FUNCTION_BLOCK FB_Generator_Random
VAR_INPUT
END_VAR
VAR_OUTPUT
END_VAR
VAR
END_VAR

END_FUNCTION_BLOCK

(* stored: Version 1.1.0.1, ProductVersion 3.1.4024.13
   POU FB_Generator_Random: Id {481933fa-f384-4460-a832-56b1a0a61ce6}, SpecialFunc None *)
